FUNCTION TFClearAllCmdModulePinza : bool
VAR_INPUT
	AspirazioneDX : POINTER TO TF_VacumOVEM;
	AspirazioneSX : POINTER TO TF_VacumOVEM;
END_VAR
VAR
END_VAR

TFOVEMClearAllCommand(AspirazioneDX^.Command);
TFOVEMClearAllCommand(AspirazioneSX^.Command);

END_FUNCTION

(* stored: Version 1.1.0.1, ProductVersion 3.1.4024.9
   POU TFClearAllCmdModulePinza: Id {a083bc3b-2742-40c4-ad3e-3fa93c56695b}, SpecialFunc None *)
